{attribute 'GeneratedUsingTerminal: EK1122-0000-0018'}
{attribute addProperty BoxType "EK1122-0000-0018"}
{attribute addProperty Id "Beckhoff_EQ2xxxsub_EK1100EK1100_AB5A94672A_0001_EQ2008_0002_0016EQ2008_D86968E311A_0002_EQ2008_0002_0017EQ2008_D86968E311A_0003_EQ2008_0002_0018EQ2008_D86968E311A_0004_EQ2008_0002_0019EQ2008_D86968E311A_0005_EQ2339_0022_0016EQ2339_0ADD710F36A_0006_EQ2339_0022_0017EQ2339_0ADD710F36A_0007_EQ2339_0022_0018EQ2339_0ADD710F36A_0008_EQ2339_0022_0019EQ2339_0ADD710F36A_0009_EQ2809_0022_0016EQ2809_E4096AA219A_0010_EQ2809_0022_0017EQ2809_E4096AA219A_0011_EQ2809_0022_0018EQ2809_E4096AA219"}
{attribute addProperty CRC "2729291093"}
{attribute addProperty Size "247"}
TYPE Beckhoff_EQ2xxxEK1122_A2ADAD55 EXTENDS EK1122_AB5A9467 :
STRUCT
	{attribute addProperty Name "Beckhoff_EQ2xxxsub_EK1100"}
	{attribute addProperty PreviousPort "Beckhoff EQ2xxxEK1122 : D"}
	Beckhoff_EQ2xxxsub_EK1100 : EK1100_AB5A9467;
	{attribute addProperty Name "A_0001_EQ2008_0002_0016"}
	{attribute addProperty PreviousPort "Beckhoff EQ2xxxsub EK1100 : C"}
	A_0001_EQ2008_0002_0016 : EQ2008_D86968E3;
	{attribute addProperty Name "A_0002_EQ2008_0002_0017"}
	{attribute addProperty PreviousPort "A_0001(EQ2008-0002-0016) : B"}
	A_0002_EQ2008_0002_0017 : EQ2008_D86968E3;
	{attribute addProperty Name "A_0003_EQ2008_0002_0018"}
	{attribute addProperty PreviousPort "A_0002(EQ2008-0002-0017) : B"}
	A_0003_EQ2008_0002_0018 : EQ2008_D86968E3;
	{attribute addProperty Name "A_0004_EQ2008_0002_0019"}
	{attribute addProperty PreviousPort "A_0003(EQ2008-0002-0018) : B"}
	A_0004_EQ2008_0002_0019 : EQ2008_D86968E3;
	{attribute addProperty Name "A_0005_EQ2339_0022_0016"}
	{attribute addProperty PreviousPort "A_0004(EQ2008-0002-0019) : B"}
	A_0005_EQ2339_0022_0016 : EQ2339_0ADD710F;
	{attribute addProperty Name "A_0006_EQ2339_0022_0017"}
	{attribute addProperty PreviousPort "A_0005(EQ2339-0022-0016) : B"}
	A_0006_EQ2339_0022_0017 : EQ2339_0ADD710F;
	{attribute addProperty Name "A_0007_EQ2339_0022_0018"}
	{attribute addProperty PreviousPort "A_0006(EQ2339-0022-0017) : B"}
	A_0007_EQ2339_0022_0018 : EQ2339_0ADD710F;
	{attribute addProperty Name "A_0008_EQ2339_0022_0019"}
	{attribute addProperty PreviousPort "A_0007(EQ2339-0022-0018) : B"}
	A_0008_EQ2339_0022_0019 : EQ2339_0ADD710F;
	{attribute addProperty Name "A_0009_EQ2809_0022_0016"}
	{attribute addProperty PreviousPort "A_0008(EQ2339-0022-0019) : B"}
	A_0009_EQ2809_0022_0016 : EQ2809_E4096AA2;
	{attribute addProperty Name "A_0010_EQ2809_0022_0017"}
	{attribute addProperty PreviousPort "A_0009(EQ2809-0022-0016) : B"}
	A_0010_EQ2809_0022_0017 : EQ2809_E4096AA2;
	{attribute addProperty Name "A_0011_EQ2809_0022_0018"}
	{attribute addProperty PreviousPort "A_0010(EQ2809-0022-0017) : B"}
	A_0011_EQ2809_0022_0018 : EQ2809_E4096AA2;
END_STRUCT
END_TYPE

(* stored: Version 1.2.0.0, ProductVersion 3.1.4024.9
   DUT Beckhoff_EQ2xxxEK1122_A2ADAD55: Id {20127d16-d99d-4fda-9164-86f279cddc36} *)
